Staubli VAL3: RobotCommandMsg.dtx

public bool bIsInitialized = true
public MessageHeader header
public RobotCommand robotCommand
public num nSerializedData
